{attribute 'qualified_only'}
VAR_GLOBAL PERSISTENT
	{attribute 'OPC.UA.DA' := '1'}
	Tags: AdsTags;
END_VAR

(* stored: Version 1.1.0.1, ProductVersion 3.1.4024.6
   GVL ADS_Standard: Id {be8f9334-fd0a-49b4-9982-0174f6f844b7} *)
